// TIA Portal V17 export
// export: Created 2024-08-20T10:59:43.0357945Z, ExportSetting WithDefaults, DisplayName Totally Integrated Automation Portal, DisplayVersion V17 Update 4, DisplayName TIA Portal Openness, DisplayVersion V17 Update 4, DisplayName TIA Portal Version Control Interface, DisplayVersion V17, DisplayName STEP 7 Professional, DisplayVersion V17 Update 4, DisplayName STEP 7 Safety, DisplayVersion V17, DisplayName WinCC Advanced, DisplayVersion V17 Update 4
DATA_BLOCK "Totalizadores"   // DB306
{ S7_Optimized_Access := 'FALSE' }
VERSION : 0.1
// stored: AutoNumber false, DBAccessibleFromOPCUA true, IsOnlyStoredInLoadMemory false, IsWriteProtectedInAS false
   VAR
      "MB-01-SO" : Int;   // Segundos em operação elevatoria principal
      "MB-01-MO" : Int;   // Minutos em operação elevatoria principal
      "MB-01-HO" : Int;   // Horas em operação elevatoria principal
      "MB-02-SO" : Int;   // Segundos em operação elevatoria principal
      "MB-02-MO" : Int;   // Minutos em operação elevatoria principal
      "MB-02-HO" : Int;   // Horas em operação elevatoria principal
      "MB-03-SO" : Int;   // Segundos em operação elevatoria principal
      "MB-03-MO" : Int;   // Minutos em operação elevatoria principal
      "MB-03-HO" : Int;   // Horas em operação elevatoria principal
      "MB-04-SO" : Int;   // Segundos em operação elevatoria principal
      "MB-04-MO" : Int;   // Minutos em operação elevatoria principal
      "MB-04-HO" : Int;   // Horas em operação elevatoria principal
   END_VAR
BEGIN
END_DATA_BLOCK
